// TIA Portal project "Project2" (V12)

(* hardware
DEVICE "S7-1200 station_1"  SIMATIC 1200-Station
   slot 0: "S7-1200 rack"  Rack  V1.0
   slot 1: "PLC_1"  CPU 1214C AC/DC/Rly  6ES7 214-1BG31-0XB0  V3.0
*)

// ===== PLC "PLC_1"  CPU 1214C AC/DC/Rly =====

DATA_BLOCK "data"   // DB1
{ S7_Optimized_Access := 'FALSE' }
VERSION : 0.1
   VAR
      contA : Int := 0;
      contB : Int := 10;
      maxValue : Int := 60;
      result : Bool := false;
      "timer" : Time := T#1000ms;
   END_VAR
BEGIN
END_DATA_BLOCK

// folder: System blocks/Program resources

DATA_BLOCK "IEC_Counter_0_DB"   // DB2
{ S7_Optimized_Access := 'FALSE' }
AUTHOR : Simatic
FAMILY : IEC
NAME : CNTR
VERSION : 1.0
// stored: InstanceOfName ?
"?"
BEGIN
END_DATA_BLOCK

DATA_BLOCK "IEC_Timer_0_DB"   // DB3
{ S7_Optimized_Access := 'FALSE' }
AUTHOR : Simatic
FAMILY : IEC
NAME : IEC_TMR
VERSION : 1.0
// stored: InstanceOfName ?
"?"
BEGIN
END_DATA_BLOCK

// folder: (top level)

ORGANIZATION_BLOCK "Main"   // OB1, LAD, ProgramCycle
TITLE = "Main Program Sweep (Cycle)"
{ S7_Optimized_Access := 'FALSE' }
VERSION : 0.1
   VAR_TEMP
      lixo : Int;
      lixo2 : Time;
   END_VAR
BEGIN

REGION Network 1
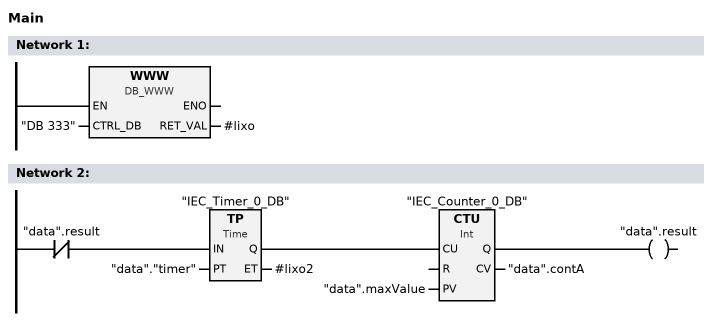
   #lixo := WWW(CTRL_DB := "DB 333");
END_REGION

REGION Network 2
   "IEC_Timer_0_DB".TP(IN := NOT "data".result, PT := "data"."timer", ET => #lixo2);
   "IEC_Counter_0_DB".CTU(CU := "IEC_Timer_0_DB".Q, PV := "data".maxValue, CV => "data".contA);
   "data".result := "IEC_Counter_0_DB".Q;
END_REGION
END_ORGANIZATION_BLOCK